TYPE TcoPlrPaletizator_Control_v_1_x_x EXTENDS TcoCore.TcoStruct:
STRUCT

		
END_STRUCT
END_TYPE

(* stored: Version 1.1.0.1
   DUT TcoPlrPaletizator_Control_v_1_x_x: Id {e80349c5-b80b-47f3-a25a-4fe537eb0b47} *)
